# EPICS IOC start-up script: iocsh/mobilellrf.iocsh
# This should be the included snippet to configure and run the deployed IOC.
# It should be loaded with
#
#   iocshLoad("$(mobilellrf_DIR)mobilellrf.iocsh", "MACRO1=xxx,MACRO2=yyy,...")

#- ###            mobilellrf ioc                    ###
#- ####################################################
#- >> Mandatory
#- ASYN_PORT1     - Asyn PORT name for agilent33220a function generator
#- ASYN_PORT2     - Asyn PORT name for arduino PLC
#- PREFIX1	  - PV PREFIX for agilent fg
#- PREFIX2	  - PV PREFIX for arduino PLC
#- PREFIX3	  - PV PREFIX for cavity selection PVs
#- IP_ADDR1	  - ethernet address of agilent fg
#- IP_ADDR2	  - ethernet address of arduino PLC
#- IOCNAME	  - Prefix for the asynRec
#- TOP	   	  - top directory for autosave
#-
#- >> Optional
#- IP_PORT1	  - IP port number for agilent fg (default 5025)
#- IP_PORT2	  - IP port number for arduino PLC (default 502)
#- DEVICE1	  - device name for agilent fg (default FUNCGEN-1)
#- DEVICE2	  - device name for arduino PLC (default ArduinoPMC:)

iocshLoad("$(agilent33220a_DIR)agilent33220a.iocsh", "IP=$(IP_ADDR1),P=$(PREFIX1),DEV=$(DEVICE1=FUNCGEN-1),ASYN_PORT=$(ASYN_PORT1)")
iocshLoad("$(arduinoplc_DIR)arduinoplc.iocsh", "IP_ADDR=$(IP_ADDR2),ASYN_PORT=$(ASYN_PORT2),TOP=$(TOP),PREFIX=$(PREFIX2),DEV_NAME=$(DEVICE2=ArduinoPMC:)")
dbLoadRecords("mobilellrf.db", "PCAV=$(PREFIX3),PRF=$(PREFIX1)$(DEVICE1=FUNCGEN-1),PLC=$(PREFIX2)$(DEVICE2=ArduinoPMC:)")
dbLoadRecords("asynRecord.db","P=$(IOCNAME),R=:asynRec,PORT=$(ASYN_PORT1),ADDR='0',IMAX='1024',OMAX='256'")
